INTERFACE ITcoScrewdriver EXTENDS __SYSTEM.IQueryInterface

METHOD Screwing : TcoCore.ITcoTaskStatus
VAR_INPUT
	ProgramNo : BYTE;
END_VAR
END_METHOD

END_INTERFACE

(* stored: Version 1.1.0.1
   Itf ITcoScrewdriver: Id {c3828ed3-c856-45da-99c0-a802bde2a9d5}
   Method Screwing: Id {2be64ce8-8445-4eb3-adaa-8ecb2d6a324d} *)
